(* IEC 61131-3 sources: AXOpen/src/core/ctrl/src/AxoComponent, 1 file *)

(* ---- AxoComponent.st ---- *)
NAMESPACE AXOpen.Core

    {S7.extern=ReadWrite}
    CLASS PUBLIC ABSTRACT AxoComponent EXTENDS AxoObject IMPLEMENTS IAxoComponent
        VAR PRIVATE
            _context    :   IAxoContext;
        END_VAR
        ///<summary>
		/// Executes the logic for manual-maintenance control.
        ///</summary>
        METHOD PUBLIC FINAL ActivateManualControl
            IF THIS._context <> NULL THEN
                 _manualControlContextCycle := _context.OpenCycleCount();
                THIS.ManualControl();
            ELSE
                _context := THIS.GetContext();
                _manualControlContextCycle := ULINT#0;        // TODO: some message should inform about this issue
            END_IF;
        END_METHOD

        ///<summary>
		/// Gets whether the AxoComponent is manually controllable.
        /// To make the AxoComponent manually controllable, it is necessary to call the `ActivateManualMode()` method cyclically.
        ///</summary>
        METHOD PUBLIC FINAL IsManuallyControllable: BOOL
           //[INLINE]THIS.CheckIfManualControlIsActivated();
            VAR
                _myContextCycleCount : ULINT;
            END_VAR
            IF THIS._context <> NULL THEN
                _myContextCycleCount := _context.OpenCycleCount();
                //When component.Service() is called "before" invoking its task _serviceContextCycle is equal to GetContext().OpenCycleCount()
                _isManuallyControllable := _manualControlContextCycle = _myContextCycleCount OR
                //When component.Service() is called "after" invoking its task (_serviceContextCycle + 1) is equal to GetContext().OpenCycleCount()
                                (_manualControlContextCycle + ULINT#1) = _myContextCycleCount;
            ELSE
                _context := THIS.GetContext();
                _isManuallyControllable := FALSE;              // TODO: some message should inform about this issue
                _myContextCycleCount := ULINT#0;
            END_IF;
                IsManuallyControllable := _isManuallyControllable;
        END_METHOD

        ///<summary>
		/// Restores this instance. This method must be implemented in derived class.
        ///</summary>
        METHOD PUBLIC ABSTRACT Restore
        END_METHOD

        ///<summary>
		/// Custom logic for manual control of the AxoComponent.
		///	This method must be implemented in derived class.
        ///</summary>
        METHOD PROTECTED ABSTRACT ManualControl
        END_METHOD

        VAR PRIVATE
           _manualControlContextCycle : ULINT;
        END_VAR

        VAR PUBLIC
            {#ix-set:AttributeName = "<#Is manually controllable#>"}
            {#ix-attr:[ReadOnly()]}
            _isManuallyControllable : BOOL;
        END_VAR

        METHOD PRIVATE CheckIfManualControlIsActivatedInlined
            VAR
                _myContextCycleCount : ULINT;
            END_VAR
            IF THIS._context <> NULL THEN
                _myContextCycleCount := _context.OpenCycleCount();
                //When component.Service() is called "before" invoking its task _serviceContextCycle is equal to GetContext().OpenCycleCount()
                _isManuallyControllable := _manualControlContextCycle = _myContextCycleCount OR
                //When component.Service() is called "after" invoking its task (_serviceContextCycle + 1) is equal to GetContext().OpenCycleCount()
                                (_manualControlContextCycle + ULINT#1) = _myContextCycleCount;
            ELSE
                _context := THIS.GetContext();
                _isManuallyControllable := FALSE;              // TODO: some message should inform about this issue
                _myContextCycleCount := ULINT#0;
            END_IF;
        END_METHOD

        METHOD PROTECTED Open
            //[INLINE]THIS.CheckIfManualControlIsActivated();
            VAR
                _myContextCycleCount : ULINT;
            END_VAR
            IF THIS._context <> NULL THEN
                _myContextCycleCount := _context.OpenCycleCount();
                //When component.Service() is called "before" invoking its task _serviceContextCycle is equal to GetContext().OpenCycleCount()
                _isManuallyControllable := _manualControlContextCycle = _myContextCycleCount OR
                //When component.Service() is called "after" invoking its task (_serviceContextCycle + 1) is equal to GetContext().OpenCycleCount()
                                (_manualControlContextCycle + ULINT#1) = _myContextCycleCount;
            ELSE
                _context := THIS.GetContext();
                _isManuallyControllable := FALSE;              // TODO: some message should inform about this issue
                _myContextCycleCount := ULINT#0;
            END_IF;
        END_METHOD

        METHOD PUBLIC Run
            THIS.Open();
            // Place the custom logic here
            THIS.Close();
        END_METHOD

        METHOD PROTECTED Close
            ;
        END_METHOD
    END_CLASS
END_NAMESPACE
